PROGRAM SprayRibRollCureSequencerSD1
VAR
	bInit : BOOL; // This sequence has been initialized.
	
	bLoading    : BOOL; // The sequence is loading tools into the bogie arms
	
	bSpraying   : BOOL; // The sequence is spraying the tools
	bRolling    : BOOL; // The sequence is rolling the tools
	bRibbing    : BOOL; // The sequence is ribbing the tools
	bCuring     : BOOL; // The sequence is curing the tools
	
	bUnloading  : BOOL; // The sequence is unloading tools from the bogie arms
	bTraversing : BOOL; // The arms are jogging.
	
	bAbleToUnload : BOOL; // TRUE when there are no part(s) blocking unload position | FALSE when there are part(s) blocking the unload position
	
END_VAR
(*
	THIS CURRENT VERSION OF THE SEQUENCER IS JUST FOR A DEMO DRY RUN WITH WX2.

	Definitions :
	Loading) We are 'Loading' until the arms have picked up the tool, and then moved them into the correct angle for spraying.
	Spraying) We are Spraying until the .NC file that is being ran by the CNC program has completed.
	Rolling) We are 'Rolling' until the .NC file that is being ran by the CNC program has completed.
	Ribbing) We are 'Ribbing' until the .NC file that is being ran by teh CNC program has competed.
	Curing) We are 'Curing' once we get into the cure position (rotation and horizontal positions) until the 'Curing timer' = 0;
	Traversing) we are considered 'moving' until we are in both the correct position with the SD jog and bogie arm rotation.
	Unloading) We are unloading until the tool has been set down, unclamped, and the arms have moved into their traverse position.
	
*)

	// These variables are for error related machine states.
VAR
	bError : BOOL;
END_VAR

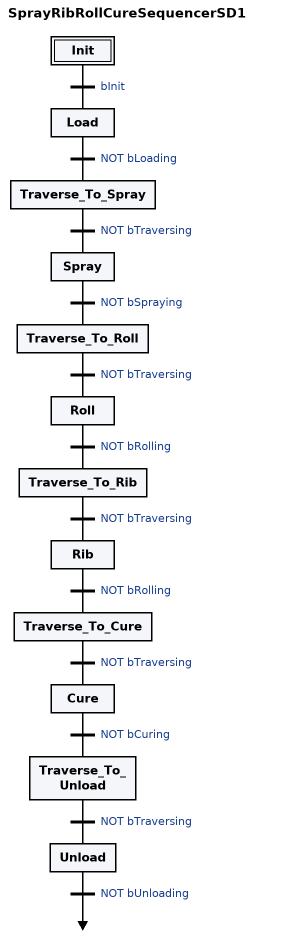
INITIAL_STEP Init:
END_STEP
TRANSITION FROM Init TO Load
    := bInit;
END_TRANSITION
STEP Load:
END_STEP
TRANSITION FROM Load TO Traverse_To_Spray
    := NOT bLoading;
END_TRANSITION
STEP Traverse_To_Spray:
END_STEP
TRANSITION FROM Traverse_To_Spray TO Spray
    := NOT bTraversing;
END_TRANSITION
STEP Spray:
END_STEP
TRANSITION FROM Spray TO Traverse_To_Roll
    := NOT bSpraying;
END_TRANSITION
STEP Traverse_To_Roll:
END_STEP
TRANSITION FROM Traverse_To_Roll TO Roll
    := NOT bTraversing;
END_TRANSITION
STEP Roll:
END_STEP
TRANSITION FROM Roll TO Traverse_To_Rib
    := NOT bRolling;
END_TRANSITION
STEP Traverse_To_Rib:
END_STEP
TRANSITION FROM Traverse_To_Rib TO Rib
    := NOT bTraversing;
END_TRANSITION
STEP Rib:
END_STEP
TRANSITION FROM Rib TO Traverse_To_Cure
    := NOT bRolling;
END_TRANSITION
STEP Traverse_To_Cure:
END_STEP
TRANSITION FROM Traverse_To_Cure TO Cure
    := NOT bTraversing;
END_TRANSITION
STEP Cure:
END_STEP
TRANSITION FROM Cure TO Traverse_To_Unload
    := NOT bCuring;
END_TRANSITION
STEP Traverse_To_Unload:
END_STEP
TRANSITION FROM Traverse_To_Unload TO Unload
    := NOT bTraversing;
END_TRANSITION
STEP Unload:
END_STEP
TRANSITION FROM Unload TO _
    := NOT bUnloading;
END_TRANSITION

END_PROGRAM

(* stored: Version 1.1.0.1, ProductVersion 3.1.4024.12
   POU SprayRibRollCureSequencerSD1: Id {4a445a81-3926-427b-8e60-b56d04d369f8}, SpecialFunc None *)
